// TIA Portal V20 export
FUNCTION_BLOCK "zPMC_Checksum"   // FB164, LAD
// stored: MemoryReserve 100, Namespace CITI_Logic, SetENOAutomatically false
   VAR_INPUT
      IN_Checksum_2 : DWord;
      IN_Checksum_3 : DWord;
      IN_Checksum_4 : DWord;
      IN_Checksum_5 : DWord;
      IN_Checksum_6 : DWord;
      IN_Checksum_7 : DWord;
      IN_Checksum_8 : DWord;
      IN_Checksum_9 : DWord;
      IN_Checksum_10 : DWord;
      IN_Checksum_11 : DWord;
      IN_Checksum_12 : DWord;
      IN_Checksum_13 : DWord;
      IN_Checksum_14 : DWord;
      IN_Checksum_15 : DWord;
      IN_Checksum_16 : DWord;
   END_VAR
   VAR_OUTPUT
      Checksum_Out : Array[1..16] of DWord;
   END_VAR
   VAR
      ON { ExternalAccessible := 'False'; ExternalVisible := 'False'; ExternalWritable := 'False'} : Bool;   // On
      OFF { ExternalAccessible := 'False'; ExternalVisible := 'False'; ExternalWritable := 'False'} : Bool;   // Off
   END_VAR
   VAR_TEMP   // added for the SCL form of the ladder/FBD networks
      _w1 : Bool;
   END_VAR
BEGIN

REGION Network 1: ==== Setup ====
   // Generate local "Always ON" and "Always OFF" conditions
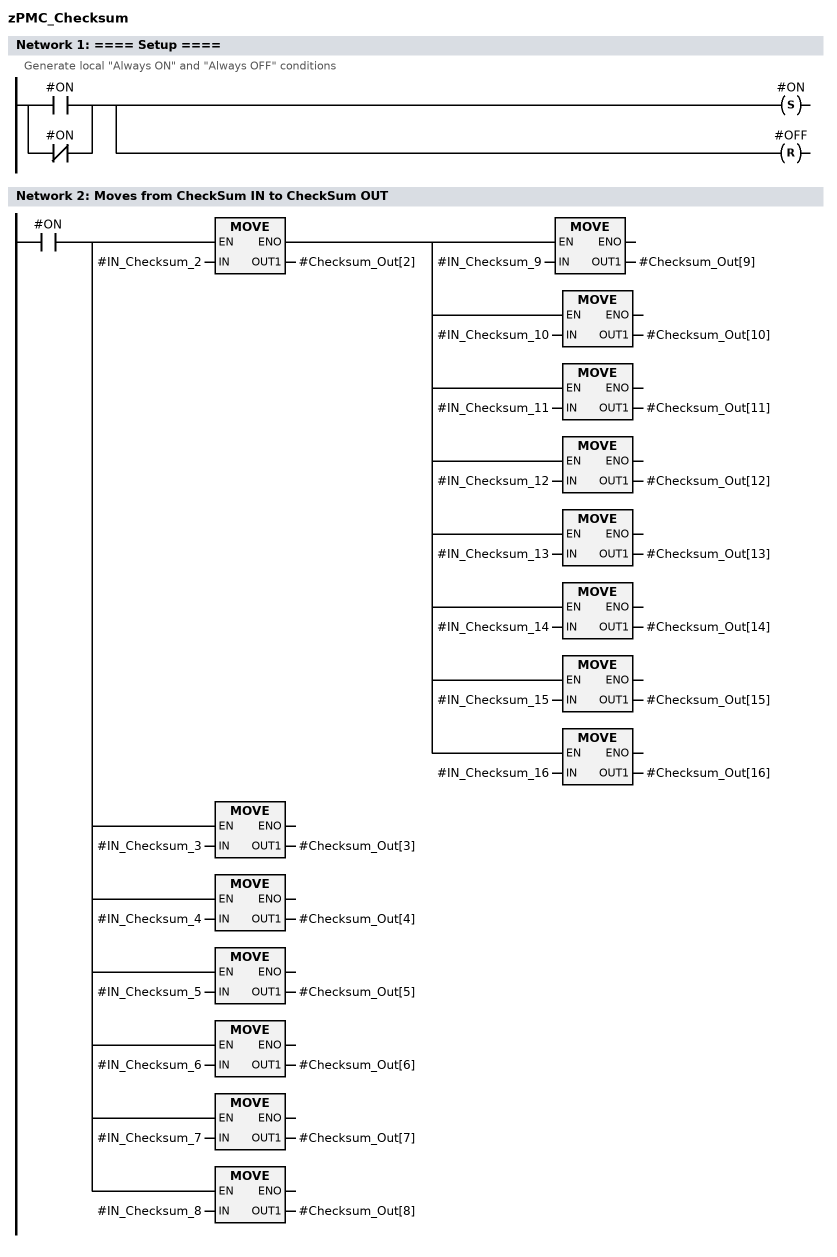
   RUNG wire#powerrail
      Contact( #ON )
      wire#w1
      S_Coil( #ON )
   END_RUNG
   RUNG wire#powerrail
      I_Contact( #ON )
   END_RUNG wire#w1
   RUNG wire#w1
      R_Coil( #OFF )
   END_RUNG
   // the same network as SCL:
   #_w1 := #ON OR NOT #ON;
   IF #_w1 THEN
       #ON := TRUE;
       #OFF := FALSE;
   END_IF;
END_REGION

REGION Network 2: Moves from CheckSum IN to CheckSum OUT
   RUNG wire#powerrail
      Contact( #ON )
      wire#w1
      { S7_GenerateENO := "TRUE" } Move(in := #IN_Checksum_2, out1 => #Checksum_Out[2])
      wire#w2
      { S7_GenerateENO := "TRUE" } Move(in := #IN_Checksum_9, out1 => #Checksum_Out[9])
   END_RUNG
   RUNG wire#w2
      { S7_GenerateENO := "TRUE" } Move(in := #IN_Checksum_10, out1 => #Checksum_Out[10])
   END_RUNG
   RUNG wire#w2
      { S7_GenerateENO := "TRUE" } Move(in := #IN_Checksum_11, out1 => #Checksum_Out[11])
   END_RUNG
   RUNG wire#w2
      { S7_GenerateENO := "TRUE" } Move(in := #IN_Checksum_12, out1 => #Checksum_Out[12])
   END_RUNG
   RUNG wire#w2
      { S7_GenerateENO := "TRUE" } Move(in := #IN_Checksum_13, out1 => #Checksum_Out[13])
   END_RUNG
   RUNG wire#w2
      { S7_GenerateENO := "TRUE" } Move(in := #IN_Checksum_14, out1 => #Checksum_Out[14])
   END_RUNG
   RUNG wire#w2
      { S7_GenerateENO := "TRUE" } Move(in := #IN_Checksum_15, out1 => #Checksum_Out[15])
   END_RUNG
   RUNG wire#w2
      { S7_GenerateENO := "TRUE" } Move(in := #IN_Checksum_16, out1 => #Checksum_Out[16])
   END_RUNG
   RUNG wire#w1
      { S7_GenerateENO := "TRUE" } Move(in := #IN_Checksum_3, out1 => #Checksum_Out[3])
   END_RUNG
   RUNG wire#w1
      { S7_GenerateENO := "TRUE" } Move(in := #IN_Checksum_4, out1 => #Checksum_Out[4])
   END_RUNG
   RUNG wire#w1
      { S7_GenerateENO := "TRUE" } Move(in := #IN_Checksum_5, out1 => #Checksum_Out[5])
   END_RUNG
   RUNG wire#w1
      { S7_GenerateENO := "TRUE" } Move(in := #IN_Checksum_6, out1 => #Checksum_Out[6])
   END_RUNG
   RUNG wire#w1
      { S7_GenerateENO := "TRUE" } Move(in := #IN_Checksum_7, out1 => #Checksum_Out[7])
   END_RUNG
   RUNG wire#w1
      { S7_GenerateENO := "TRUE" } Move(in := #IN_Checksum_8, out1 => #Checksum_Out[8])
   END_RUNG
   // the same network as SCL:
   // ENO of a box is taken as its EN; it also drops when the box reports an error
   IF #ON THEN
       #Checksum_Out[2] := #IN_Checksum_2;
       #Checksum_Out[9] := #IN_Checksum_9;
       #Checksum_Out[10] := #IN_Checksum_10;
       #Checksum_Out[11] := #IN_Checksum_11;
       #Checksum_Out[12] := #IN_Checksum_12;
       #Checksum_Out[13] := #IN_Checksum_13;
       #Checksum_Out[14] := #IN_Checksum_14;
       #Checksum_Out[15] := #IN_Checksum_15;
       #Checksum_Out[16] := #IN_Checksum_16;
       #Checksum_Out[3] := #IN_Checksum_3;
       #Checksum_Out[4] := #IN_Checksum_4;
       #Checksum_Out[5] := #IN_Checksum_5;
       #Checksum_Out[6] := #IN_Checksum_6;
       #Checksum_Out[7] := #IN_Checksum_7;
       #Checksum_Out[8] := #IN_Checksum_8;
   END_IF;
END_REGION
END_FUNCTION_BLOCK
